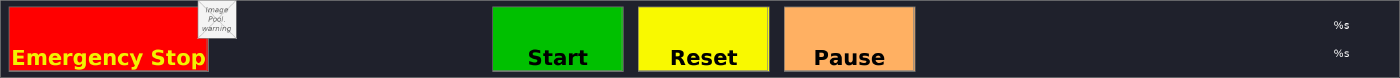
VISUALIZATION FOOTER  // 1920x108
    Rectangle (0,0 1920x108)
    Rectangle (1760,0 160x108), text variable: MAIN.fb_TimeStamp.SystemTime
    Textfield (1760,20 160x30), "%s", text variable: MAIN.fb_TimeStamp.SystemTime
    Textfield (1760,59 160x30), "%s", text variable: MAIN.fb_TimeStamp.SystemDate
    Button (675,9 180x90), "Start"
        tap IO_HMI.bStart p3779583253=TRUE
    Button (1075,9 180x90), "Pause"
        tap IO_HMI.bStop
    Button (875,9 180x90), "Reset"
        tap IO_HMI.bReset
    Button (12,9 274x90), "Emergency Stop"
        OnMouseClick: toggle IO_HMI.bEstop
    Image (271,0 53x53), invisible if: IO_control.bEstop, image: ImagePool.warning
END_VISUALIZATION

(* stored: Version 1.1.0.1, ProductVersion 3.1.4024.12
   Visu FOOTER: Id {1ad4d962-13b7-46d6-8df4-1a0acdd38e9c} *)
